{attribute 'qualified_only'}
VAR_GLOBAL
	VERSION			: STRING := '2.0.0';
	IsReset 		: BOOL := TRUE;
	IsTestProject 	: BOOL := TRUE;
	IsRunning 		: BOOL;
	TestPointer 	: POINTER TO BOOL; //For 32/64bit check
	IsTc2 			: BOOL := FALSE;
END_VAR

(* stored: Version 1.1.0.1, ProductVersion 3.1.4024.12
   GVL GVL_AdsClientTests: Id {df176121-69f2-4834-ba42-2f401dc63f8f} *)
